PROGRAM MAIN
VAR
	
     fbRedColor 		: FB_RedColor;
	 fbBlueColor 		: FB_BlueColor;
	 
	 fbSquareRed 		: FB_Square(Color:= fbRedColor );
	 fbSquareBlue 		: FB_Square(Color:= fbBlueColor );
	 
	 fbCircleRed 		: FB_Circle(Color:= fbRedColor );
	 fbCircleBlue 		: FB_Circle(Color:= fbBlueColor );
	 
	 bstartDemo1		: BOOL;
	 
END_VAR

IF bstartDemo1 THEN
	bstartDemo1 := FALSE;
	
	fbSquareRed.Draw();
	fbSquareBlue.Draw();
	
	fbCircleRed.Draw();
	fbCircleBlue.Draw();
	
END_IF

END_PROGRAM

(* stored: Version 1.1.0.1, ProductVersion 3.1.4024.12
   POU MAIN: Id {1392cc94-1c79-40f6-929c-7566d1e6cfbf}, SpecialFunc None *)
